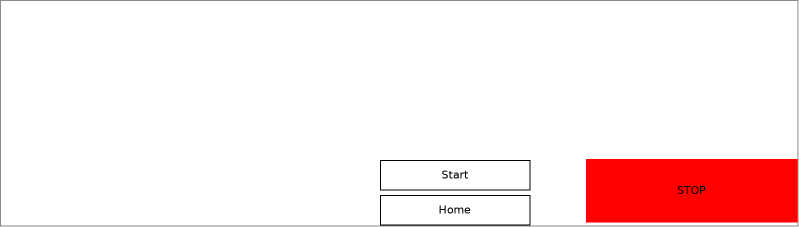
VISUALIZATION Homing  // 799x227
    Rectangle (380,195 150x30), "Home"
        tap INIT.bHome
    Rectangle (380,160 150x30), "Start", colour toggle: INIT.bEN
        toggle INIT.bENCouple
    Rectangle (586,159 211x63), "STOP", colour toggle: GVL.StopALL
        toggle GVL.StopALL
END_VISUALIZATION

(* stored: Version 1.1.0.1, ProductVersion 3.1.4022.17
   Visu Homing: Id {64b99297-7dc5-4d27-8bf3-5813020828b3} *)
